// TIA Portal V17 export
// export: Created 2022-02-03T14:45:12.1424825Z, ExportSetting WithDefaults, DisplayName Totally Integrated Automation Portal, DisplayVersion V17, DisplayName TIA Portal Openness, DisplayVersion V17, DisplayName TIA Portal Version Control Interface, DisplayVersion V17, DisplayName SINAMICS Startdrive Advanced, DisplayVersion V17, DisplayName SINAMICS Startdrive G130, G150, S120, S150, SINAMICS MV, S210, DisplayVersion V17, DisplayName SINAMICS Startdrive G110M, G120, G120C, G120D, G120P, G115D, DisplayVersion V17, DisplayName STEP 7 Professional, DisplayVersion V17, DisplayName STEP 7 Safety, DisplayVersion V17, DisplayName WinCC Advanced, DisplayVersion V17
ORGANIZATION_BLOCK "CyclicInterruptWeight"   // OB30, LAD, CyclicInterrupt
VERSION : 0.1
// stored: AutoNumber true, IsIECCheckEnabled false, SetENOAutomatically false
   VAR_INPUT
      Initial_Call : Bool;   // Initial call of this OB
      Event_Count : Int;   // Events discarded
   END_VAR
   VAR_TEMP
      tempWeight : Real;
   END_VAR
BEGIN

REGION Network 1
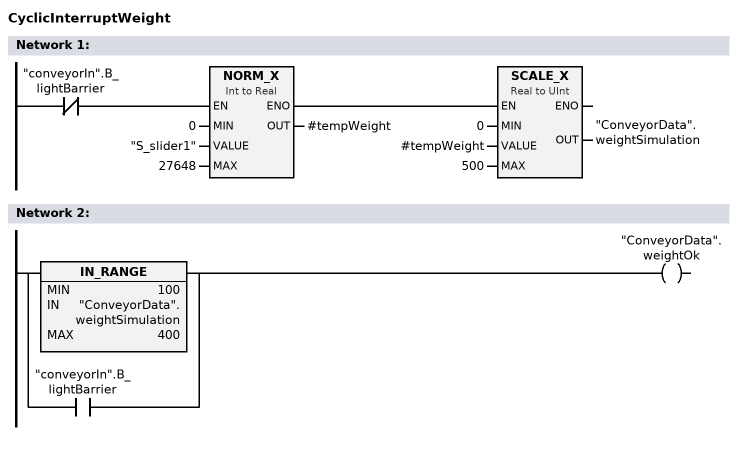
   RUNG wire#powerrail
      I_Contact( "conveyorIn".B_lightBarrier )
      { S7_Templates := "[SrcType := Int, DestType := Real]" } Normalize(min := 0, value := "S_slider1", max := 27648, out => #tempWeight)
      { S7_Templates := "[SrcType := Real, DestType := UInt]" } Scale(min := 0, value := #tempWeight, max := 500, out => "ConveyorData".weightSimulation)
   END_RUNG
   // the same network as SCL:
   IF NOT "conveyorIn".B_lightBarrier THEN
       #tempWeight := NORM_X(MIN := 0, VALUE := "S_slider1", MAX := 27648);
       "ConveyorData".weightSimulation := SCALE_X(MIN := 0, VALUE := #tempWeight, MAX := 500);
   END_IF;
END_REGION

REGION Network 2
   RUNG wire#powerrail
      { S7_Templates := "SrcType := UInt" } InRange(min := 100, in := "ConveyorData".weightSimulation, max := 400)
      wire#w1
      Coil( "ConveyorData".weightOk )
   END_RUNG
   RUNG wire#powerrail
      Contact( "conveyorIn".B_lightBarrier )
   END_RUNG wire#w1
   // the same network as SCL:
   "ConveyorData".weightOk := ((100 <= "ConveyorData".weightSimulation) AND ("ConveyorData".weightSimulation <= 400)) OR "conveyorIn".B_lightBarrier;
END_REGION
END_ORGANIZATION_BLOCK
